// TIA Portal V19 export
TYPE "LSNTP_typeDiagnostics"
TITLE = typeDiagnostics
// Provides a structure for detailed diagnostics
// stored: Access Published
   STRUCT
      status { ExternalVisible := 'False'; ExternalWritable := 'False'} : Word;   // Status of the block or error identification when error occurred
      subfunctionStatus { ExternalVisible := 'False'; ExternalWritable := 'False'} : DWord;   // Status or return value of called FBs, FCs and system blocks
      stateNumber { ExternalVisible := 'False'; ExternalWritable := 'False'} : DInt;   // State in the state machine of the block where the error occurred
   END_STRUCT;
END_TYPE
